FUNCTION_BLOCK Muxi (* Basic Function Block Type *)
  (* Standard: 61499-2 *)
  (* Version 0.0, 6/8/2016, Andrei, nxtControl GmbH, Template *)
  PACKAGE Main;
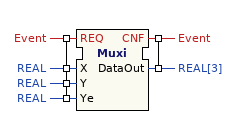
  EVENT_INPUT
    REQ WITH X, Y, Ye; (* Normal Execution Request *)
  END_EVENT
  EVENT_OUTPUT
    CNF WITH DataOut; (* Execution Confirmation *)
  END_EVENT
  VAR_INPUT
    X : REAL; (* Input event qualifier *)
    Y : REAL;
    Ye : REAL;
  END_VAR
  VAR_OUTPUT
    DataOut : ARRAY [0..2] OF REAL; (* Output event qualifier *)
  END_VAR
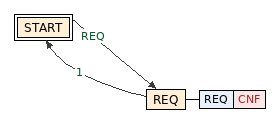
  EC_STATES
    START; (* Initial State *)
    REQ : REQ -> CNF; (* Normal execution *)
  END_STATES
  EC_TRANSITIONS
    START TO REQ := REQ;
    REQ TO START := 1;
  END_TRANSITIONS
  ALGORITHM REQ IN ST: (* Normally executed algorithm *)
DataOut[0] := X;
DataOut[1] := Y;
DataOut[2] := Ye;
  END_ALGORITHM
END_FUNCTION_BLOCK
